// TIA Portal V17 export
// export: Created 2025-03-07T09:17:17.166723Z, ExportSetting WithDefaults, DisplayName Totally Integrated Automation Portal, DisplayVersion V17 Update 8, DisplayName TIA Portal Openness, DisplayVersion V17 Update 8, DisplayName TIA Portal Version Control Interface, DisplayVersion V17, DisplayName SINAMICS Startdrive Advanced, DisplayVersion V17 SP2, DisplayName SINAMICS Startdrive G110M, G120, G120C, G120D, G120P, G115D, DisplayVersion V17 SP2, DisplayName SINAMICS Startdrive G130, G150, S120, S150, SINAMICS MV, S210, DisplayVersion V17 SP2, DisplayName STEP 7 Professional, DisplayVersion V17 Update 8, DisplayName SINUMERIK ONE STEP 7 Toolbox, DisplayVersion V17 Update 12, DisplayName SINUMERIK 840D sl STEP 7 Toolbox, DisplayVersion V17 Update 12, DisplayName STEP 7 Safety, DisplayVersion V17 Update 6, DisplayName WinCC Advanced, DisplayVersion V17 Update 8
DATA_BLOCK "DB353_M_UNIT_01_STA_4"   // DB353
{ S7_Optimized_Access := 'FALSE'; DB_Accessible_From_OPC_UA := 'FALSE' }
AUTHOR : ETXETAR
VERSION : 1.0
// stored: AutoNumber false, DBAccessibleFromOPCUA false, DBAccessibleFromWebserver true, IsOnlyStoredInLoadMemory false, IsWriteProtectedInAS false
   VAR RETAIN
      M_CODES_UNIT_01_STA_4 : "M_FUNCTIONS_UNIT_STATION_4";
   END_VAR
BEGIN
   // M_CODES_UNIT_01_STA_4.M170 : M170- ADVANCE Z14 (READ-IN DISABLE)
   // M_CODES_UNIT_01_STA_4.Ack_M170 : ACKNOWLEDGE M170- ADVANCE Z14 (READ-IN DISABLE)
   // M_CODES_UNIT_01_STA_4.M171 : M171- RETURN Z14 (READ-IN DISABLE)
   // M_CODES_UNIT_01_STA_4.Ack_M171 : ACKNOWLEDGE M171- RETURN Z14 (READ-IN DISABLE)
END_DATA_BLOCK
